//{attribute 'qualified_only'}
//{attribute 'strict'}
{attribute 'to_string'}
TYPE E_PackagingState :
(
	Idle,
    Moving,
    Sealing,
    Error

);
END_TYPE

(* stored: Version 1.1.0.1
   DUT E_PackagingState: Id {ad63989a-1d27-4069-8f6b-6479bb59c5a9} *)
